LIN {X 0,Y 1.29,Z 1190.871,A -85,B 0,C 180,E1 -4317.069,E2 -4317.069} C_VEL
LIN {X 0,Y 1.294,Z 1190.864,A -85,B 0,C 180,E1 -4142.963,E2 -4142.963} C_VEL
LIN {X 0,Y 0.337,Z 1190.89,A -85,B 0,C 180,E1 -3965.753,E2 -3965.753} C_VEL
LIN {X 0,Y 2.354,Z 1192.89,A -85,B 0,C 180,E1 -3956.562,E2 -3956.562} C_VEL
LIN {X 0,Y 2.354,Z 1215,A -85,B 0,C 180,E1 -3956.562,E2 -3956.562} C_VEL
LIN {X 0,Y 2.354,Z 1215,A -85,B 0,C 180,E1 -3956.562,E2 -3956.562}

QRS_NEXT_CUT()

QRS_NEXT()
QRS_HOME()

END
